TYPE ST145_Recipe_t :
STRUCT
    xUseVerLeft  : BOOL; // Is the left vertical picker element is used
    xUseVerRight : BOOL; // Is the right vertical picker element is used
    FeederConfig : FeederDelays_t;
END_STRUCT
END_TYPE

(* stored: Version 1.1.0.1, ProductVersion 3.1.4024.6
   DUT ST145_Recipe_t: Id {0bf075a3-3e7c-4472-bcff-87e2f1141a83} *)
